// TIA Portal V15.1 export
// export: Created 2020-06-12T07:35:54.9599609Z, ExportSetting None, DisplayName Totally Integrated Automation Portal, DisplayVersion V15.1, DisplayName TIA Portal Openness, DisplayVersion V15.1, DisplayName STEP 7 Professional, DisplayVersion V15.1, DisplayName STEP 7 Safety, DisplayVersion V15.1, DisplayName WinCC Advanced, DisplayVersion V15.1
FUNCTION "Desk_ES1GD03" : Void   // FC165, FBD
{ S7_Optimized_Access := 'TRUE' }
// stored: SetENOAutomatically False
BEGIN

REGION Network 1: ES1GD03 SPB: Desk is on
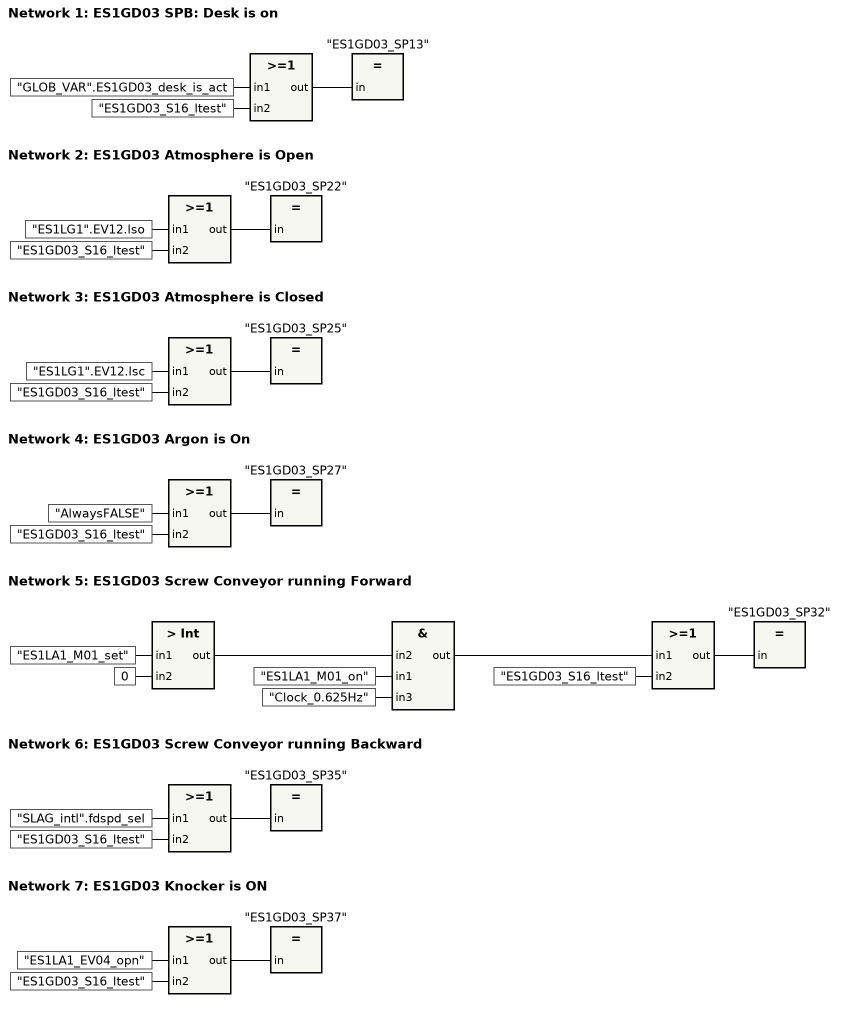
   "ES1GD03_SP13" := "GLOB_VAR".ES1GD03_desk_is_act OR "ES1GD03_S16_ltest";
END_REGION

REGION Network 2: ES1GD03 Atmosphere is Open
   "ES1GD03_SP22" := "ES1LG1".EV12.lso OR "ES1GD03_S16_ltest";
END_REGION

REGION Network 3: ES1GD03 Atmosphere is Closed
   "ES1GD03_SP25" := "ES1LG1".EV12.lsc OR "ES1GD03_S16_ltest";
END_REGION

REGION Network 4: ES1GD03 Argon is On
   "ES1GD03_SP27" := "AlwaysFALSE" OR "ES1GD03_S16_ltest";
END_REGION

REGION Network 5: ES1GD03 Screw Conveyor running Forward
   "ES1GD03_SP32" := (("ES1LA1_M01_set" > 0) AND "ES1LA1_M01_on" AND "Clock_0.625Hz") OR "ES1GD03_S16_ltest";
END_REGION

REGION Network 6: ES1GD03 Screw Conveyor running Backward
   // There is vibro-feeder, no backward command.
   "ES1GD03_SP35" := "SLAG_intl".fdspd_sel OR "ES1GD03_S16_ltest";
END_REGION

REGION Network 7: ES1GD03 Knocker is ON
   "ES1GD03_SP37" := "ES1LA1_EV04_opn" OR "ES1GD03_S16_ltest";
END_REGION
END_FUNCTION
